// TIA Portal V20 export
DATA_BLOCK "DB_Manual"   // DB21
// stored: Access Published, MemoryReserve 100, Namespace LineD1
   VAR
      Conveyor : Struct
         ID : Int;
         Enable : Bool;
         Run : Bool;
         in : Bool;
      END_STRUCT;
      Line : Struct
         D1 : Struct
            Conveyor { S7_SetPoint := 'True'} : Array[_.minD1.._.maxD1] of "LineD1.ManualInputs";
         END_STRUCT;
      END_STRUCT;
   END_VAR
BEGIN
END_DATA_BLOCK
